Staubli VAL3: serverCmd.pgx

program serverCmd()
  local bool bFlag
  local num nArgs[8]
  local num nBuffer[30]
  local num nBytes
  local num nIndex
  local num nNbArgs
  local num ni
  local string sBuffer
  local string sCommand
begin
  //server task - read and write on socket
  //SETUP - CLEAR BUFFER
  clearBuffer(sSocket1)
  ////////FOREVER LOOP - TASK////////
  while (true)
    //nBytes = number of bytes read to nBuffer
    //nBytes must be less than 30 and not empty
    nBytes=sioGet(sSocket1,nBuffer)
    if (nBytes>0) and (nBytes<30)
      //INPUT PARSING
      call argumentParse(nBuffer,nBytes,nArgs,nNbArgs,sBuffer,sCommand)
      //CHECK COMMAND
      call commandCheck(nArgs,nNbArgs,sBuffer,sCommand,bFlag)
      if bFlag==true
        //EXECUTE COMMAND
        call commandExecute(nArgs,nNbArgs,sBuffer,sCommand)
      else
        logMsg("serverCmd: bFlag == false")
      endIf
      //OUTPUT WRITE
      call socketWrite(sBuffer,nBuffer)
      nBytes=sioSet(sSocket1,nBuffer)
      if (nBytes<0)
        logMsg("serverCmd: sioSet error > "+toString("",nBytes))
      endIf
    else
      logMsg("serverCmd: sioget error > "+chr(nBytes))
    endIf
  endWhile
end
